   1:  PR[91,3] = PR[90,3] + 65.195;
   1:L PR[91] R[100]mm/sec CNT100;
   1:  PR[91,1] = PR[90,1] + -66.038;
   1:  PR[91,2] = PR[90,2] + 18.167;
   1:  PR[91,3] = PR[90,3] + 63.911;
   1:L PR[91] R[100]mm/sec CNT100;
   1:  PR[91,1] = PR[90,1] + -70.511;
   1:  PR[91,2] = PR[90,2] + 15.205;
   1:L PR[91] R[100]mm/sec CNT100;
   1:  PR[91,1] = PR[90,1] + -74.081;
   1:  PR[91,2] = PR[90,2] + 11.663;
   1:  PR[91,3] = PR[90,3] + 63.930;
   1:L PR[91] R[100]mm/sec CNT100;
   1:  PR[91,1] = PR[90,1] + -76.653;
   1:  PR[91,2] = PR[90,2] + 7.733;
   1:  PR[91,3] = PR[90,3] + 63.947;
   1:L PR[91] R[100]mm/sec CNT100;
   1:  PR[91,1] = PR[90,1] + -78.198;
   1:  PR[91,2] = PR[90,2] + 3.559;
   1:  PR[91,3] = PR[90,3] + 63.964;
   1:L PR[91] R[100]mm/sec CNT100;
   1:  PR[91,1] = PR[90,1] + -78.594;
   1:  PR[91,2] = PR[90,2] + 0.279;
   1:  PR[91,3] = PR[90,3] + 63.979;
   1:L PR[91] R[100]mm/sec CNT100;
   1:  PR[91,1] = PR[90,1] + -78.770;
   1:  PR[91,2] = PR[90,2] + -0.700;
   1:  PR[91,3] = PR[90,3] + 63.991;
   1:L PR[91] R[100]mm/sec CNT100;
   1:  PR[91,1] = PR[90,1] + -78.578;
   1:  PR[91,2] = PR[90,2] + -1.617;
   1:  PR[91,3] = PR[90,3] + 63.994;
   1:L PR[91] R[100]mm/sec CNT100;
   1:  PR[91,1] = PR[90,1] + -78.140;
   1:  PR[91,2] = PR[90,2] + -5.208;
   1:  PR[91,3] = PR[90,3] + 63.998;
   1:L PR[91] R[100]mm/sec CNT100;
   1:  PR[91,1] = PR[90,1] + -77.858;
   1:  PR[91,2] = PR[90,2] + -5.991;
   1:  PR[91,3] = PR[90,3] + 64.010;
   1:L PR[91] R[100]mm/sec CNT100;
   1:  PR[91,1] = PR[90,1] + -76.508;
   1:  PR[91,2] = PR[90,2] + -9.566;
   1:  PR[91,3] = PR[90,3] + 64.013;
   1:L PR[91] R[100]mm/sec CNT100;
   1:  PR[91,1] = PR[90,1] + -76.251;
   1:  PR[91,2] = PR[90,2] + -9.971;
   1:  PR[91,3] = PR[90,3] + 64.027;
   1:L PR[91] R[100]mm/sec CNT100;
   1:  PR[91,1] = PR[90,1] + -73.777;
   1:  PR[91,2] = PR[90,2] + -13.651;
   1:  PR[91,3] = PR[90,3] + 64.028;
   1:L PR[91] R[100]mm/sec CNT100;
   1:  PR[91,1] = PR[90,1] + -73.531;
   1:  PR[91,2] = PR[90,2] + -13.889;
   1:  PR[91,3] = PR[90,3] + 64.044;
   1:L PR[91] R[100]mm/sec CNT100;
   1:  PR[91,1] = PR[90,1] + -69.827;
   1:  PR[91,2] = PR[90,2] + -17.193;
   1:  PR[91,3] = PR[90,3] + 64.045;
   1:L PR[91] R[100]mm/sec CNT100;
   1:  PR[91,1] = PR[90,1] + -68.494;
   1:  PR[91,2] = PR[90,2] + -17.992;
   1:  PR[91,3] = PR[90,3] + 64.062;
   1:L PR[91] R[100]mm/sec CNT100;
   1:  PR[91,1] = PR[90,1] + -64.853;
   1:  PR[91,2] = PR[90,2] + -20.132;
   1:  PR[91,3] = PR[90,3] + 64.068;
   1:L PR[91] R[100]mm/sec CNT100;
   1:  PR[91,1] = PR[90,1] + -60.373;
   1:  PR[91,2] = PR[90,2] + -21.812;
   1:  PR[91,3] = PR[90,3] + 64.083;
   1:L PR[91] R[100]mm/sec CNT100;
   1:  PR[91,1] = PR[90,1] + -59.088;
   1:  PR[91,2] = PR[90,2] + -22.281;
   1:  PR[91,3] = PR[90,3] + 64.099;
   1:L PR[91] R[100]mm/sec CNT100;
   1:  PR[91,1] = PR[90,1] + -52.980;
   1:  PR[91,2] = PR[90,2] + -23.447;
   1:  PR[91,3] = PR[90,3] + 64.104;
   1:L PR[91] R[100]mm/sec CNT100;
   1:  PR[91,1] = PR[90,1] + -50.323;
   1:  PR[91,2] = PR[90,2] + -23.702;
   1:  PR[91,3] = PR[90,3] + 64.126;
   1:L PR[91] R[100]mm/sec CNT100;
   1:  PR[91,1] = PR[90,1] + -47.192;
   1:  PR[91,2] = PR[90,2] + -23.829;
   1:  PR[91,3] = PR[90,3] + 64.135;
   1:L PR[91] R[100]mm/sec CNT100;
   1:  PR[91,1] = PR[90,1] + -43.588;
   1:  PR[91,2] = PR[90,2] + -23.669;
   1:  PR[91,3] = PR[90,3] + 64.146;
   1:L PR[91] R[100]mm/sec CNT100;
   1:  PR[91,1] = PR[90,1] + -41.498;
   1:  PR[91,2] = PR[90,2] + -23.638;
   1:  PR[91,3] = PR[90,3] + 64.159;
   1:L PR[91] R[100]mm/sec CNT100;
   1:  PR[91,1] = PR[90,1] + -39.473;
   1:  PR[91,2] = PR[90,2] + -23.516;
   1:  PR[91,3] = PR[90,3] + 64.166;
   1:L PR[91] R[100]mm/sec CNT100;
   1:  PR[91,1] = PR[90,1] + -36.086;
   1:  PR[91,2] = PR[90,2] + -23.043;
   1:  PR[91,3] = PR[90,3] + 64.173;
   1:L PR[91] R[100]mm/sec CNT100;
   1:  PR[91,1] = PR[90,1] + -32.879;
   1:  PR[91,2] = PR[90,2] + -22.411;
   1:  PR[91,3] = PR[90,3] + 64.185;
   1:L PR[91] R[100]mm/sec CNT100;
   1:  PR[91,1] = PR[90,1] + -29.442;
   1:  PR[91,2] = PR[90,2] + -21.943;
   1:  PR[91,3] = PR[90,3] + 64.197;
   1:L PR[91] R[100]mm/sec CNT100;
   1:  PR[91,1] = PR[90,1] + -23.128;
   1:  PR[91,2] = PR[90,2] + -20.482;
   1:  PR[91,3] = PR[90,3] + 64.209;
   1:L PR[91] R[100]mm/sec CNT100;
   1:  PR[91,1] = PR[90,1] + -19.496;
   1:  PR[91,2] = PR[90,2] + -22.048;
   1:  PR[91,3] = PR[90,3] + 64.231;
   1:L PR[91] R[100]mm/sec CNT100;
   1:  PR[91,1] = PR[90,1] + -17.322;
   1:  PR[91,2] = PR[90,2] + -22.682;
   1:  PR[91,3] = PR[90,3] + 64.245;
   1:L PR[91] R[100]mm/sec CNT100;
   1:  PR[91,1] = PR[90,1] + -14.113;
   1:  PR[91,2] = PR[90,2] + -23.536;
   1:  PR[91,3] = PR[90,3] + 64.253;
   1:L PR[91] R[100]mm/sec CNT100;
   1:  PR[91,1] = PR[90,1] + -8.398;
   1:  PR[91,2] = PR[90,2] + -23.980;
   1:  PR[91,3] = PR[90,3] + 64.265;
   1:L PR[91] R[100]mm/sec CNT100;
   1:  PR[91,1] = PR[90,1] + -2.492;
   1:  PR[91,2] = PR[90,2] + -23.372;
   1:  PR[91,3] = PR[90,3] + 64.285;
   1:L PR[91] R[100]mm/sec CNT100;
   1:  PR[91,1] = PR[90,1] + -0.519;
   1:  PR[91,2] = PR[90,2] + -22.811;
   1:  PR[91,3] = PR[90,3] + 64.306;
   1:L PR[91] R[100]mm/sec CNT100;
   1:  PR[91,1] = PR[90,1] + 3.330;
   1:  PR[91,2] = PR[90,2] + -21.668;
   1:  PR[91,3] = PR[90,3] + 64.313;
   1:L PR[91] R[100]mm/sec CNT100;
   1:  PR[91,1] = PR[90,1] + 6.156;
   1:  PR[91,2] = PR[90,2] + -20.297;
   1:  PR[91,3] = PR[90,3] + 64.327;
   1:L PR[91] R[100]mm/sec CNT100;
   1:  PR[91,1] = PR[90,1] + 11.934;
   1:  PR[91,2] = PR[90,2] + -23.385;
   1:  PR[91,3] = PR[90,3] + 64.338;
   1:L PR[91] R[100]mm/sec CNT100;
   1:  PR[91,1] = PR[90,1] + 17.314;
   1:  PR[91,2] = PR[90,2] + -24.854;
   1:  PR[91,3] = PR[90,3] + 64.361;
   1:L PR[91] R[100]mm/sec CNT100;
   1:  PR[91,1] = PR[90,1] + 22.909;
   1:  PR[91,2] = PR[90,2] + -25.082;
   1:  PR[91,3] = PR[90,3] + 64.380;
   1:L PR[91] R[100]mm/sec CNT100;
   1:  PR[91,1] = PR[90,1] + 28.505;
   1:  PR[91,2] = PR[90,2] + -24.027;
   1:  PR[91,3] = PR[90,3] + 64.400;
   1:L PR[91] R[100]mm/sec CNT100;
   1:  PR[91,1] = PR[90,1] + 29.696;
   1:  PR[91,2] = PR[90,2] + -23.650;
   1:  PR[91,3] = PR[90,3] + 64.420;
   1:L PR[91] R[100]mm/sec CNT100;
   1:  PR[91,1] = PR[90,1] + 33.478;
   1:  PR[91,2] = PR[90,2] + -24.727;
   1:  PR[91,3] = PR[90,3] + 64.424;
   1:L PR[91] R[100]mm/sec CNT100;
   1:  PR[91,1] = PR[90,1] + 35.307;
   1:  PR[91,2] = PR[90,2] + -25.218;
   1:  PR[91,3] = PR[90,3] + 64.438;
   1:L PR[91] R[100]mm/sec CNT100;
   1:  PR[91,1] = PR[90,1] + 41.330;
   1:  PR[91,2] = PR[90,2] + -25.987;
   1:  PR[91,3] = PR[90,3] + 64.445;
   1:L PR[91] R[100]mm/sec CNT100;
   1:  PR[91,1] = PR[90,1] + 45.575;
   1:  PR[91,2] = PR[90,2] + -26.004;
   1:  PR[91,3] = PR[90,3] + 64.466;
   1:L PR[91] R[100]mm/sec CNT100;
   1:  PR[91,1] = PR[90,1] + 46.620;
   1:  PR[91,2] = PR[90,2] + -26.023;
   1:  PR[91,3] = PR[90,3] + 64.481;
   1:L PR[91] R[100]mm/sec CNT100;
   1:  PR[91,1] = PR[90,1] + 49.214;
   1:  PR[91,2] = PR[90,2] + -25.837;
   1:  PR[91,3] = PR[90,3] + 64.485;
   1:L PR[91] R[100]mm/sec CNT100;
   1:  PR[91,1] = PR[90,1] + 51.095;
   1:  PR[91,2] = PR[90,2] + -25.664;
   1:  PR[91,3] = PR[90,3] + 64.494;
   1:L PR[91] R[100]mm/sec CNT100;
   1:  PR[91,1] = PR[90,1] + 56.435;
   1:  PR[91,2] = PR[90,2] + -24.677;
   1:  PR[91,3] = PR[90,3] + 64.500;
   1:L PR[91] R[100]mm/sec CNT100;
   1:  PR[91,1] = PR[90,1] + 63.147;
   1:  PR[91,2] = PR[90,2] + -22.494;
   1:  PR[91,3] = PR[90,3] + 64.519;
   1:L PR[91] R[100]mm/sec CNT100;
   1:  PR[91,1] = PR[90,1] + 63.555;
   1:  PR[91,2] = PR[90,2] + -22.305;
   1:  PR[91,3] = PR[90,3] + 64.544;
   1:L PR[91] R[100]mm/sec CNT100;
   1:  PR[91,1] = PR[90,1] + 65.028;
   1:  PR[91,2] = PR[90,2] + -21.507;
   1:  PR[91,3] = PR[90,3] + 64.546;
   1:L PR[91] R[100]mm/sec CNT100;
   1:  PR[91,1] = PR[90,1] + 69.095;
   1:  PR[91,2] = PR[90,2] + -19.132;
   1:  PR[91,3] = PR[90,3] + 64.551;
   1:L PR[91] R[100]mm/sec CNT100;
   1:  PR[91,1] = PR[90,1] + 71.773;
   1:  PR[91,2] = PR[90,2] + -16.745;
   1:  PR[91,3] = PR[90,3] + 64.568;
   1:L PR[91] R[100]mm/sec CNT100;
   1:  PR[91,1] = PR[90,1] + 73.617;
   1:  PR[91,2] = PR[90,2] + -15.079;
   1:  PR[91,3] = PR[90,3] + 64.580;
   1:L PR[91] R[100]mm/sec CNT100;
   1:  PR[91,1] = PR[90,1] + 76.861;
   1:  PR[91,2] = PR[90,2] + -10.536;
   1:  PR[91,3] = PR[90,3] + 64.589;
   1:L PR[91] R[100]mm/sec CNT100;
   1:  PR[91,1] = PR[90,1] + 78.802;
   1:  PR[91,2] = PR[90,2] + -5.697;
   1:  PR[91,3] = PR[90,3] + 64.609;
   1:L PR[91] R[100]mm/sec CNT100;
   1:  PR[91,1] = PR[90,1] + 79.399;
   1:  PR[91,2] = PR[90,2] + -1.168;
   1:  PR[91,3] = PR[90,3] + 64.627;
   1:L PR[91] R[100]mm/sec CNT100;
   1:  PR[91,1] = PR[90,1] + 79.474;
   1:  PR[91,2] = PR[90,2] + -0.700;
   1:  PR[91,3] = PR[90,3] + 64.643;
   1:L PR[91] R[100]mm/sec CNT100;
   1:  PR[91,1] = PR[90,1] + 78.963;
   1:  PR[91,2] = PR[90,2] + 3.215;
   1:  PR[91,3] = PR[90,3] + 64.645;
   1:L PR[91] R[100]mm/sec CNT100;
   1:  PR[91,1] = PR[90,1] + 78.903;
   1:  PR[91,2] = PR[90,2] + 3.455;
   1:  PR[91,3] = PR[90,3] + 64.658;
   1:L PR[91] R[100]mm/sec CNT100;
   1:  PR[91,1] = PR[90,1] + 78.799;
   1:  PR[91,2] = PR[90,2] + 4.246;
   1:  PR[91,3] = PR[90,3] + 64.659;
   1:L PR[91] R[100]mm/sec CNT100;
   1:  PR[91,1] = PR[90,1] + 76.856;
   1:  PR[91,2] = PR[90,2] + 9.086;
   1:  PR[91,3] = PR[90,3] + 64.662;
   1:L PR[91] R[100]mm/sec CNT100;
   1:  PR[91,1] = PR[90,1] + 73.613;
   1:  PR[91,2] = PR[90,2] + 13.624;
   1:  PR[91,3] = PR[90,3] + 64.680;
   1:L PR[91] R[100]mm/sec CNT100;
   1:  PR[91,1] = PR[90,1] + 69.094;
   1:  PR[91,2] = PR[90,2] + 17.673;
   1:  PR[91,3] = PR[90,3] + 64.700;
   1:L PR[91] R[100]mm/sec CNT100;
   1:  PR[91,1] = PR[90,1] + 65.028;
   1:  PR[91,2] = PR[90,2] + 20.050;
   1:  PR[91,3] = PR[90,3] + 64.721;
   1:L PR[91] R[100]mm/sec CNT100;
   1:  PR[91,1] = PR[90,1] + 63.571;
   1:  PR[91,2] = PR[90,2] + 20.840;
   1:  PR[91,3] = PR[90,3] + 64.738;
   1:L PR[91] R[100]mm/sec CNT100;
   1:  PR[91,1] = PR[90,1] + 63.168;
   1:  PR[91,2] = PR[90,2] + 21.026;
   1:  PR[91,3] = PR[90,3] + 64.743;
   1:L PR[91] R[100]mm/sec CNT100;
   1:  PR[91,1] = PR[90,1] + 56.445;
   1:  PR[91,2] = PR[90,2] + 23.216;
   1:  PR[91,3] = PR[90,3] + 64.745;
   1:L PR[91] R[100]mm/sec CNT100;
   1:  PR[91,1] = PR[90,1] + 51.095;
   1:  PR[91,2] = PR[90,2] + 24.206;
   1:  PR[91,3] = PR[90,3] + 64.770;
   1:L PR[91] R[100]mm/sec CNT100;
   1:  PR[91,1] = PR[90,1] + 49.215;
   1:  PR[91,2] = PR[90,2] + 24.378;
   1:  PR[91,3] = PR[90,3] + 64.789;
   1:L PR[91] R[100]mm/sec CNT100;
   1:  PR[91,1] = PR[90,1] + 46.620;
   1:  PR[91,2] = PR[90,2] + 24.564;
   1:  PR[91,3] = PR[90,3] + 64.795;
   1:L PR[91] R[100]mm/sec CNT100;
   1:  PR[91,1] = PR[90,1] + 45.575;
   1:  PR[91,2] = PR[90,2] + 24.545;
   1:  PR[91,3] = PR[90,3] + 64.804;
   1:L PR[91] R[100]mm/sec CNT100;
   1:  PR[91,1] = PR[90,1] + 41.330;
   1:  PR[91,2] = PR[90,2] + 24.528;
   1:  PR[91,3] = PR[90,3] + 64.808;
   1:L PR[91] R[100]mm/sec CNT100;
   1:  PR[91,1] = PR[90,1] + 35.307;
   1:  PR[91,2] = PR[90,2] + 23.759;
   1:  PR[91,3] = PR[90,3] + 64.823;
   1:L PR[91] R[100]mm/sec CNT100;
   1:  PR[91,1] = PR[90,1] + 33.478;
   1:  PR[91,2] = PR[90,2] + 23.268;
   1:  PR[91,3] = PR[90,3] + 64.844;
   1:L PR[91] R[100]mm/sec CNT100;
   1:  PR[91,1] = PR[90,1] + 29.686;
   1:  PR[91,2] = PR[90,2] + 22.188;
   1:  PR[91,3] = PR[90,3] + 64.851;
   1:L PR[91] R[100]mm/sec CNT100;
   1:  PR[91,1] = PR[90,1] + 28.655;
   1:  PR[91,2] = PR[90,2] + 22.526;
   1:  PR[91,3] = PR[90,3] + 64.865;
   1:L PR[91] R[100]mm/sec CNT100;
   1:  PR[91,1] = PR[90,1] + 27.759;
   1:  PR[91,2] = PR[90,2] + 22.715;
   1:  PR[91,3] = PR[90,3] + 64.868;
   1:L PR[91] R[100]mm/sec CNT100;
   1:  PR[91,1] = PR[90,1] + 22.910;
   1:  PR[91,2] = PR[90,2] + 23.623;
   1:  PR[91,3] = PR[90,3] + 64.872;
   1:L PR[91] R[100]mm/sec CNT100;
   1:  PR[91,1] = PR[90,1] + 17.313;
   1:  PR[91,2] = PR[90,2] + 23.395;
   1:  PR[91,3] = PR[90,3] + 64.889;
   1:L PR[91] R[100]mm/sec CNT100;
   1:  PR[91,1] = PR[90,1] + 11.931;
   1:  PR[91,2] = PR[90,2] + 21.925;
   1:  PR[91,3] = PR[90,3] + 64.909;
   1:L PR[91] R[100]mm/sec CNT100;
   1:  PR[91,1] = PR[90,1] + 6.142;
   1:  PR[91,2] = PR[90,2] + 18.842;
   1:  PR[91,3] = PR[90,3] + 64.928;
   1:L PR[91] R[100]mm/sec CNT100;
   1:  PR[91,1] = PR[90,1] + 4.093;
   1:  PR[91,2] = PR[90,2] + 19.856;
   1:  PR[91,3] = PR[90,3] + 64.951;
   1:L PR[91] R[100]mm/sec CNT100;
   1:  PR[91,1] = PR[90,1] + 3.348;
   1:  PR[91,2] = PR[90,2] + 20.203;
   1:  PR[91,3] = PR[90,3] + 64.959;
   1:L PR[91] R[100]mm/sec CNT100;
   1:  PR[91,1] = PR[90,1] + -0.515;
   1:  PR[91,2] = PR[90,2] + 21.353;
   1:  PR[91,3] = PR[90,3] + 64.962;
   1:L PR[91] R[100]mm/sec CNT100;
   1:  PR[91,1] = PR[90,1] + -2.470;
   1:  PR[91,2] = PR[90,2] + 21.909;
   1:  PR[91,3] = PR[90,3] + 64.976;
   1:L PR[91] R[100]mm/sec CNT100;
   1:  PR[91,1] = PR[90,1] + -8.387;
   1:  PR[91,2] = PR[90,2] + 22.521;
   1:  PR[91,3] = PR[90,3] + 64.983;
   1:L PR[91] R[100]mm/sec CNT100;
   1:  PR[91,1] = PR[90,1] + -14.097;
   1:  PR[91,2] = PR[90,2] + 22.080;
   1:  PR[91,3] = PR[90,3] + 65.004;
   1:L PR[91] R[100]mm/sec CNT100;
   1:  PR[91,1] = PR[90,1] + -17.311;
   1:  PR[91,2] = PR[90,2] + 21.224;
   1:  PR[91,3] = PR[90,3] + 65.024;
   1:L PR[91] R[100]mm/sec CNT100;
   1:  PR[91,1] = PR[90,1] + -19.480;
   1:  PR[91,2] = PR[90,2] + 20.596;
   1:  PR[91,3] = PR[90,3] + 65.036;
   1:L PR[91] R[100]mm/sec CNT100;
   1:  PR[91,1] = PR[90,1] + -23.127;
   1:  PR[91,2] = PR[90,2] + 19.024;
   1:  PR[91,3] = PR[90,3] + 65.044;
   1:L PR[91] R[100]mm/sec CNT100;
   1:  PR[91,1] = PR[90,1] + -29.591;
   1:  PR[91,2] = PR[90,2] + 20.509;
   1:  PR[91,3] = PR[90,3] + 65.057;
   1:L PR[91] R[100]mm/sec CNT100;
   1:  PR[91,1] = PR[90,1] + -31.869;
   1:  PR[91,2] = PR[90,2] + 20.801;
   1:  PR[91,3] = PR[90,3] + 65.081;
   1:L PR[91] R[100]mm/sec CNT100;
   1:  PR[91,1] = PR[90,1] + -36.385;
   1:  PR[91,2] = PR[90,2] + 21.658;
   1:  PR[91,3] = PR[90,3] + 65.089;
   1:L PR[91] R[100]mm/sec CNT100;
   1:  PR[91,1] = PR[90,1] + -41.380;
   1:  PR[91,2] = PR[90,2] + 22.076;
   1:  PR[91,3] = PR[90,3] + 65.105;
   1:L PR[91] R[100]mm/sec CNT100;
   1:  PR[91,1] = PR[90,1] + -42.819;
   1:  PR[91,2] = PR[90,2] + 22.268;
   1:  PR[91,3] = PR[90,3] + 65.122;
   1:L PR[91] R[100]mm/sec CNT100;
   1:  PR[91,1] = PR[90,1] + -44.055;
   1:  PR[91,2] = PR[90,2] + 22.365;
   1:  PR[91,3] = PR[90,3] + 65.127;
   1:L PR[91] R[100]mm/sec CNT100;
   1:  PR[91,1] = PR[90,1] + -47.939;
   1:  PR[91,2] = PR[90,2] + 22.299;
   1:  PR[91,3] = PR[90,3] + 65.132;
   1:L PR[91] R[100]mm/sec CNT100;
   1:  PR[91,1] = PR[90,1] + -53.378;
   1:  PR[91,2] = PR[90,2] + 21.968;
   1:  PR[91,3] = PR[90,3] + 65.145;
   1:L PR[91] R[100]mm/sec CNT100;
   1:  PR[91,1] = PR[90,1] + -57.549;
   1:  PR[91,2] = PR[90,2] + 21.084;
   1:  PR[91,3] = PR[90,3] + 65.164;
   1:L PR[91] R[100]mm/sec CNT100;
   1:  PR[91,1] = PR[90,1] + -60.125;
   1:  PR[91,2] = PR[90,2] + 20.512;
   1:  PR[91,3] = PR[90,3] + 65.179;
   1:L PR[91] R[100]mm/sec CNT100;
   1:  PR[91,1] = PR[90,1] + -61.822;
   1:  PR[91,2] = PR[90,2] + 19.851;
   1:  PR[91,3] = PR[90,3] + 65.189;
   1:L PR[91] R[100]mm/sec CNT100;
   1:  PR[91] = PR[90];
   1:  PR[91,1] = PR[90,1] + -64.918;
   1:  PR[91,2] = PR[90,2] + 18.355;
   1:  PR[91,3] = PR[90,3] + 66.495;
   1:L PR[91] R[100]mm/sec CNT100;
   1:  PR[91,1] = PR[90,1] + -67.688;
   1:  PR[91,2] = PR[90,2] + 16.655;
   1:  PR[91,3] = PR[90,3] + 65.208;
   1:L PR[91] R[100]mm/sec CNT100;
   1:  PR[91,1] = PR[90,1] + -69.669;
   1:  PR[91,2] = PR[90,2] + 15.342;
   1:  PR[91,3] = PR[90,3] + 65.220;
   1:L PR[91] R[100]mm/sec CNT100;
   1:  PR[91,1] = PR[90,1] + -73.276;
   1:  PR[91,2] = PR[90,2] + 11.769;
   1:  PR[91,3] = PR[90,3] + 65.228;
   1:L PR[91] R[100]mm/sec CNT100;
   1:  PR[91,1] = PR[90,1] + -75.873;
   1:  PR[91,2] = PR[90,2] + 7.805;
   1:  PR[91,3] = PR[90,3] + 65.246;
   1:L PR[91] R[100]mm/sec CNT100;
   1:  PR[91,1] = PR[90,1] + -77.433;
   1:  PR[91,2] = PR[90,2] + 3.596;
   1:  PR[91,3] = PR[90,3] + 65.263;
   1:L PR[91] R[100]mm/sec CNT100;
   1:  PR[91,1] = PR[90,1] + -77.752;
   1:  PR[91,2] = PR[90,2] + 0.956;
   1:  PR[91,3] = PR[90,3] + 65.279;
   1:L PR[91] R[100]mm/sec CNT100;
   1:  PR[91,1] = PR[90,1] + -78.050;
   1:  PR[91,2] = PR[90,2] + -0.700;
   1:  PR[91,3] = PR[90,3] + 65.288;
   1:L PR[91] R[100]mm/sec CNT100;
   1:  PR[91,1] = PR[90,1] + -77.966;
   1:  PR[91,2] = PR[90,2] + -1.098;
   1:  PR[91,3] = PR[90,3] + 65.294;
   1:L PR[91] R[100]mm/sec CNT100;
   1:  PR[91,1] = PR[90,1] + -77.460;
   1:  PR[91,2] = PR[90,2] + -5.248;
   1:  PR[91,3] = PR[90,3] + 65.295;
   1:L PR[91] R[100]mm/sec CNT100;
   1:  PR[91,1] = PR[90,1] + -75.804;
   1:  PR[91,2] = PR[90,2] + -9.653;
   1:  PR[91,3] = PR[90,3] + 65.310;
   1:L PR[91] R[100]mm/sec CNT100;
   1:  PR[91,1] = PR[90,1] + -75.073;
   1:  PR[91,2] = PR[90,2] + -10.749;
   1:  PR[91,3] = PR[90,3] + 65.327;
   1:L PR[91] R[100]mm/sec CNT100;
   1:  PR[91,1] = PR[90,1] + -72.949;
   1:  PR[91,2] = PR[90,2] + -13.691;
   1:  PR[91,3] = PR[90,3] + 65.331;
   1:L PR[91] R[100]mm/sec CNT100;
   1:  PR[91,1] = PR[90,1] + -68.910;
   1:  PR[91,2] = PR[90,2] + -17.302;
   1:  PR[91,3] = PR[90,3] + 65.344;
   1:L PR[91] R[100]mm/sec CNT100;
   1:  PR[91,1] = PR[90,1] + -66.512;
   1:  PR[91,2] = PR[90,2] + -18.739;
   1:  PR[91,3] = PR[90,3] + 65.363;
   1:L PR[91] R[100]mm/sec CNT100;
   1:  PR[91,1] = PR[90,1] + -63.913;
   1:  PR[91,2] = PR[90,2] + -20.268;
   1:  PR[91,3] = PR[90,3] + 65.373;
   1:L PR[91] R[100]mm/sec CNT100;
   1:  PR[91,1] = PR[90,1] + -58.107;
   1:  PR[91,2] = PR[90,2] + -22.444;
   1:  PR[91,3] = PR[90,3] + 65.384;
   1:L PR[91] R[100]mm/sec CNT100;
   1:  PR[91,1] = PR[90,1] + -52.157;
   1:  PR[91,2] = PR[90,2] + -23.581;
   1:  PR[91,3] = PR[90,3] + 65.406;
   1:L PR[91] R[100]mm/sec CNT100;
   1:  PR[91,1] = PR[90,1] + -47.855;
   1:  PR[91,2] = PR[90,2] + -23.994;
   1:  PR[91,3] = PR[90,3] + 65.427;
   1:L PR[91] R[100]mm/sec CNT100;
   1:  PR[91,1] = PR[90,1] + -46.414;
   1:  PR[91,2] = PR[90,2] + -24.052;
   1:  PR[91,3] = PR[90,3] + 65.443;
   1:L PR[91] R[100]mm/sec CNT100;
   1:  PR[91,1] = PR[90,1] + -44.701;
   1:  PR[91,2] = PR[90,2] + -23.976;
   1:  PR[91,3] = PR[90,3] + 65.448;
   1:L PR[91] R[100]mm/sec CNT100;
   1:  PR[91,1] = PR[90,1] + -40.730;
   1:  PR[91,2] = PR[90,2] + -23.917;
   1:  PR[91,3] = PR[90,3] + 65.454;
   1:L PR[91] R[100]mm/sec CNT100;
   1:  PR[91,1] = PR[90,1] + -36.785;
   1:  PR[91,2] = PR[90,2] + -23.680;
   1:  PR[91,3] = PR[90,3] + 65.468;
   1:L PR[91] R[100]mm/sec CNT100;
   1:  PR[91,1] = PR[90,1] + -35.256;
   1:  PR[91,2] = PR[90,2] + -23.467;
   1:  PR[91,3] = PR[90,3] + 65.482;
   1:L PR[91] R[100]mm/sec CNT100;
   1:  PR[91,1] = PR[90,1] + -33.740;
   1:  PR[91,2] = PR[90,2] + -23.168;
   1:  PR[91,3] = PR[90,3] + 65.487;
   1:L PR[91] R[100]mm/sec CNT100;
   1:  PR[91,1] = PR[90,1] + -27.820;
   1:  PR[91,2] = PR[90,2] + -22.362;
   1:  PR[91,3] = PR[90,3] + 65.493;
   1:L PR[91] R[100]mm/sec CNT100;
   1:  PR[91,1] = PR[90,1] + -24.290;
   1:  PR[91,2] = PR[90,2] + -21.549;
   1:  PR[91,3] = PR[90,3] + 65.514;
   1:L PR[91] R[100]mm/sec CNT100;
   1:  PR[91,1] = PR[90,1] + -21.649;
   1:  PR[91,2] = PR[90,2] + -21.053;
   1:  PR[91,3] = PR[90,3] + 65.526;
   1:L PR[91] R[100]mm/sec CNT100;
   1:  PR[91,1] = PR[90,1] + -18.816;
   1:  PR[91,2] = PR[90,2] + -22.269;
   1:  PR[91,3] = PR[90,3] + 65.536;
   1:L PR[91] R[100]mm/sec CNT100;
   1:  PR[91,1] = PR[90,1] + -17.201;
   1:  PR[91,2] = PR[90,2] + -22.739;
   1:  PR[91,3] = PR[90,3] + 65.547;
   1:L PR[91] R[100]mm/sec CNT100;
   1:  PR[91,1] = PR[90,1] + -13.448;
   1:  PR[91,2] = PR[90,2] + -23.739;
   1:  PR[91,3] = PR[90,3] + 65.553;
   1:L PR[91] R[100]mm/sec CNT100;
   1:  PR[91,1] = PR[90,1] + -7.645;
   1:  PR[91,2] = PR[90,2] + -24.196;
   1:  PR[91,3] = PR[90,3] + 65.567;
   1:L PR[91] R[100]mm/sec CNT100;
   1:  PR[91,1] = PR[90,1] + -6.885;
   1:  PR[91,2] = PR[90,2] + -24.130;
   1:  PR[91,3] = PR[90,3] + 65.587;
   1:L PR[91] R[100]mm/sec CNT100;
   1:  PR[91,1] = PR[90,1] + -1.660;
   1:  PR[91,2] = PR[90,2] + -23.602;
   1:  PR[91,3] = PR[90,3] + 65.590;
   1:L PR[91] R[100]mm/sec CNT100;
   1:  PR[91,1] = PR[90,1] + 1.593;
   1:  PR[91,2] = PR[90,2] + -22.676;
   1:  PR[91,3] = PR[90,3] + 65.608;
   1:L PR[91] R[100]mm/sec CNT100;
   1:  PR[91,1] = PR[90,1] + 4.238;
   1:  PR[91,2] = PR[90,2] + -21.891;
   1:  PR[91,3] = PR[90,3] + 65.620;
   1:L PR[91] R[100]mm/sec CNT100;
   1:  PR[91,1] = PR[90,1] + 6.446;
   1:  PR[91,2] = PR[90,2] + -20.820;
   1:  PR[91,3] = PR[90,3] + 65.630;
   1:L PR[91] R[100]mm/sec CNT100;
   1:  PR[91,1] = PR[90,1] + 10.926;
   1:  PR[91,2] = PR[90,2] + -23.208;
   1:  PR[91,3] = PR[90,3] + 65.639;
   1:L PR[91] R[100]mm/sec CNT100;
   1:  PR[91,1] = PR[90,1] + 11.742;
   1:  PR[91,2] = PR[90,2] + -23.583;
   1:  PR[91,3] = PR[90,3] + 65.657;
   1:L PR[91] R[100]mm/sec CNT100;
   1:  PR[91,1] = PR[90,1] + 17.142;
   1:  PR[91,2] = PR[90,2] + -25.054;
   1:  PR[91,3] = PR[90,3] + 65.660;
   1:L PR[91] R[100]mm/sec CNT100;
   1:  PR[91,1] = PR[90,1] + 17.170;
   1:  PR[91,2] = PR[90,2] + -25.060;
   1:  PR[91,3] = PR[90,3] + 65.680;
   1:L PR[91] R[100]mm/sec CNT100;
   1:  PR[91,1] = PR[90,1] + 22.787;
   1:  PR[91,2] = PR[90,2] + -25.287;
   1:L PR[91] R[100]mm/sec CNT100;
   1:  PR[91,1] = PR[90,1] + 28.397;
   1:  PR[91,2] = PR[90,2] + -24.234;
   1:  PR[91,3] = PR[90,3] + 65.700;
   1:L PR[91] R[100]mm/sec CNT100;
   1:  PR[91,1] = PR[90,1] + 29.133;
   1:  PR[91,2] = PR[90,2] + -24.016;
   1:  PR[91,3] = PR[90,3] + 65.720;
   1:L PR[91] R[100]mm/sec CNT100;
   1:  PR[91,1] = PR[90,1] + 32.821;
   1:  PR[91,2] = PR[90,2] + -25.060;
   1:  PR[91,3] = PR[90,3] + 65.722;
   1:L PR[91] R[100]mm/sec CNT100;
   1:  PR[91,1] = PR[90,1] + 34.276;
   1:  PR[91,2] = PR[90,2] + -25.447;
   1:  PR[91,3] = PR[90,3] + 65.736;
   1:L PR[91] R[100]mm/sec CNT100;
   1:  PR[91,1] = PR[90,1] + 40.204;
   1:  PR[91,2] = PR[90,2] + -26.207;
   1:  PR[91,3] = PR[90,3] + 65.741;
   1:L PR[91] R[100]mm/sec CNT100;
   1:  PR[91,1] = PR[90,1] + 45.797;
   1:  PR[91,2] = PR[90,2] + -26.222;
   1:  PR[91,3] = PR[90,3] + 65.762;
   1:L PR[91] R[100]mm/sec CNT100;
   1:  PR[91,1] = PR[90,1] + 46.538;
   1:  PR[91,2] = PR[90,2] + -26.133;
   1:  PR[91,3] = PR[90,3] + 65.782;
   1:L PR[91] R[100]mm/sec CNT100;
   1:  PR[91,1] = PR[90,1] + 50.425;
   1:  PR[91,2] = PR[90,2] + -25.777;
   1:  PR[91,3] = PR[90,3] + 65.785;
   1:L PR[91] R[100]mm/sec CNT100;
   1:  PR[91,1] = PR[90,1] + 55.385;
   1:  PR[91,2] = PR[90,2] + -24.854;
   1:  PR[91,3] = PR[90,3] + 65.799;
   1:L PR[91] R[100]mm/sec CNT100;
   1:  PR[91,1] = PR[90,1] + 61.784;
   1:  PR[91,2] = PR[90,2] + -22.774;
   1:  PR[91,3] = PR[90,3] + 65.816;
   1:L PR[91] R[100]mm/sec CNT100;
   1:  PR[91,1] = PR[90,1] + 62.965;
   1:  PR[91,2] = PR[90,2] + -22.228;
   1:  PR[91,3] = PR[90,3] + 65.840;
   1:L PR[91] R[100]mm/sec CNT100;
   1:  PR[91,1] = PR[90,1] + 66.536;
   1:  PR[91,2] = PR[90,2] + -20.295;
   1:  PR[91,3] = PR[90,3] + 65.845;
   1:L PR[91] R[100]mm/sec CNT100;
   1:  PR[91,1] = PR[90,1] + 68.202;
   1:  PR[91,2] = PR[90,2] + -19.322;
   1:  PR[91,3] = PR[90,3] + 65.859;
   1:L PR[91] R[100]mm/sec CNT100;
   1:  PR[91,1] = PR[90,1] + 72.782;
   1:  PR[91,2] = PR[90,2] + -15.222;
   1:  PR[91,3] = PR[90,3] + 65.866;
   1:L PR[91] R[100]mm/sec CNT100;
   1:  PR[91,1] = PR[90,1] + 76.061;
   1:  PR[91,2] = PR[90,2] + -10.636;
   1:  PR[91,3] = PR[90,3] + 65.888;
   1:L PR[91] R[100]mm/sec CNT100;
   1:  PR[91,1] = PR[90,1] + 78.023;
   1:  PR[91,2] = PR[90,2] + -5.748;
   1:  PR[91,3] = PR[90,3] + 65.908;
   1:L PR[91] R[100]mm/sec CNT100;
   1:  PR[91,1] = PR[90,1] + 78.523;
   1:  PR[91,2] = PR[90,2] + -1.956;
   1:  PR[91,3] = PR[90,3] + 65.926;
   1:L PR[91] R[100]mm/sec CNT100;
   1:  PR[91,1] = PR[90,1] + 78.725;
   1:  PR[91,2] = PR[90,2] + -0.700;
   1:  PR[91,3] = PR[90,3] + 65.940;
   1:L PR[91] R[100]mm/sec CNT100;
   1:  PR[91,1] = PR[90,1] + 78.326;
   1:  PR[91,2] = PR[90,2] + 2.359;
   1:  PR[91,3] = PR[90,3] + 65.944;
   1:L PR[91] R[100]mm/sec CNT100;
   1:  PR[91,1] = PR[90,1] + 78.218;
   1:  PR[91,2] = PR[90,2] + 2.785;
   1:  PR[91,3] = PR[90,3] + 65.955;
   1:L PR[91] R[100]mm/sec CNT100;
   1:  PR[91,1] = PR[90,1] + 78.021;
   1:  PR[91,2] = PR[90,2] + 4.296;
   1:  PR[91,3] = PR[90,3] + 65.957;
   1:L PR[91] R[100]mm/sec CNT100;
   1:  PR[91,1] = PR[90,1] + 76.057;
   1:  PR[91,2] = PR[90,2] + 9.183;
   1:  PR[91,3] = PR[90,3] + 65.962;
   1:L PR[91] R[100]mm/sec CNT100;
   1:  PR[91,1] = PR[90,1] + 72.779;
   1:  PR[91,2] = PR[90,2] + 13.767;
   1:  PR[91,3] = PR[90,3] + 65.981;
   1:L PR[91] R[100]mm/sec CNT100;
   1:  PR[91,1] = PR[90,1] + 68.210;
   1:  PR[91,2] = PR[90,2] + 17.857;
   1:  PR[91,3] = PR[90,3] + 66.001;
   1:L PR[91] R[100]mm/sec CNT100;
   1:  PR[91,1] = PR[90,1] + 66.535;
   1:  PR[91,2] = PR[90,2] + 18.836;
   1:  PR[91,3] = PR[90,3] + 66.022;
   1:L PR[91] R[100]mm/sec CNT100;
   1:  PR[91,1] = PR[90,1] + 62.978;
   1:  PR[91,2] = PR[90,2] + 20.764;
   1:  PR[91,3] = PR[90,3] + 66.029;
   1:L PR[91] R[100]mm/sec CNT100;
   1:  PR[91,1] = PR[90,1] + 61.800;
   1:  PR[91,2] = PR[90,2] + 21.308;
   1:  PR[91,3] = PR[90,3] + 66.043;
   1:L PR[91] R[100]mm/sec CNT100;
   1:  PR[91,1] = PR[90,1] + 55.390;
   1:  PR[91,2] = PR[90,2] + 23.394;
   1:  PR[91,3] = PR[90,3] + 66.048;
   1:L PR[91] R[100]mm/sec CNT100;
   1:  PR[91,1] = PR[90,1] + 50.424;
   1:  PR[91,2] = PR[90,2] + 24.318;
   1:  PR[91,3] = PR[90,3] + 66.072;
   1:L PR[91] R[100]mm/sec CNT100;
   1:  PR[91,1] = PR[90,1] + 46.538;
   1:  PR[91,2] = PR[90,2] + 24.674;
   1:  PR[91,3] = PR[90,3] + 66.090;
   1:L PR[91] R[100]mm/sec CNT100;
   1:  PR[91,1] = PR[90,1] + 45.797;
   1:  PR[91,2] = PR[90,2] + 24.763;
   1:  PR[91,3] = PR[90,3] + 66.103;
   1:L PR[91] R[100]mm/sec CNT100;
   1:  PR[91,1] = PR[90,1] + 40.204;
   1:  PR[91,2] = PR[90,2] + 24.749;
   1:  PR[91,3] = PR[90,3] + 66.106;
   1:L PR[91] R[100]mm/sec CNT100;
   1:  PR[91,1] = PR[90,1] + 34.276;
   1:  PR[91,2] = PR[90,2] + 23.988;
   1:  PR[91,3] = PR[90,3] + 66.126;
   1:L PR[91] R[100]mm/sec CNT100;
   1:  PR[91,1] = PR[90,1] + 32.821;
   1:  PR[91,2] = PR[90,2] + 23.601;
   1:  PR[91,3] = PR[90,3] + 66.147;
   1:L PR[91] R[100]mm/sec CNT100;
   1:  PR[91,1] = PR[90,1] + 29.186;
   1:  PR[91,2] = PR[90,2] + 22.572;
   1:  PR[91,3] = PR[90,3] + 66.152;
   1:L PR[91] R[100]mm/sec CNT100;
   1:  PR[91,1] = PR[90,1] + 28.119;
   1:  PR[91,2] = PR[90,2] + 22.830;
   1:  PR[91,3] = PR[90,3] + 66.166;
   1:L PR[91] R[100]mm/sec CNT100;
   1:  PR[91,1] = PR[90,1] + 22.787;
   1:  PR[91,2] = PR[90,2] + 23.828;
   1:  PR[91,3] = PR[90,3] + 66.170;
   1:L PR[91] R[100]mm/sec CNT100;
   1:  PR[91,1] = PR[90,1] + 17.169;
   1:  PR[91,2] = PR[90,2] + 23.601;
   1:  PR[91,3] = PR[90,3] + 66.189;
   1:L PR[91] R[100]mm/sec CNT100;
   1:  PR[91,1] = PR[90,1] + 17.141;
   1:  PR[91,2] = PR[90,2] + 23.595;
   1:  PR[91,3] = PR[90,3] + 66.209;
   1:L PR[91] R[100]mm/sec CNT100;
   1:  PR[91,1] = PR[90,1] + 11.740;
   1:  PR[91,2] = PR[90,2] + 22.123;
   1:L PR[91] R[100]mm/sec CNT100;
   1:  PR[91,1] = PR[90,1] + 10.925;
   1:  PR[91,2] = PR[90,2] + 21.749;
   1:  PR[91,3] = PR[90,3] + 66.228;
   1:L PR[91] R[100]mm/sec CNT100;
   1:  PR[91,1] = PR[90,1] + 6.439;
   1:  PR[91,2] = PR[90,2] + 19.396;
   1:  PR[91,3] = PR[90,3] + 66.232;
   1:L PR[91] R[100]mm/sec CNT100;
   1:  PR[91,1] = PR[90,1] + 4.247;
   1:  PR[91,2] = PR[90,2] + 20.429;
   1:  PR[91,3] = PR[90,3] + 66.250;
   1:L PR[91] R[100]mm/sec CNT100;
   1:  PR[91,1] = PR[90,1] + 1.585;
   1:  PR[91,2] = PR[90,2] + 21.221;
   1:  PR[91,3] = PR[90,3] + 66.258;
   1:L PR[91] R[100]mm/sec CNT100;
   1:  PR[91,1] = PR[90,1] + -1.634;
   1:  PR[91,2] = PR[90,2] + 22.138;
   1:  PR[91,3] = PR[90,3] + 66.268;
   1:L PR[91] R[100]mm/sec CNT100;
   1:  PR[91,1] = PR[90,1] + -6.863;
   1:  PR[91,2] = PR[90,2] + 22.669;
   1:  PR[91,3] = PR[90,3] + 66.280;
   1:L PR[91] R[100]mm/sec CNT100;
   1:  PR[91,1] = PR[90,1] + -7.633;
   1:  PR[91,2] = PR[90,2] + 22.737;
   1:  PR[91,3] = PR[90,3] + 66.298;
   1:L PR[91] R[100]mm/sec CNT100;
   1:  PR[91,1] = PR[90,1] + -13.436;
   1:  PR[91,2] = PR[90,2] + 22.282;
   1:  PR[91,3] = PR[90,3] + 66.301;
   1:L PR[91] R[100]mm/sec CNT100;
   1:  PR[91,1] = PR[90,1] + -17.195;
   1:  PR[91,2] = PR[90,2] + 21.281;
   1:  PR[91,3] = PR[90,3] + 66.322;
   1:L PR[91] R[100]mm/sec CNT100;
   1:  PR[91,1] = PR[90,1] + -18.805;
   1:  PR[91,2] = PR[90,2] + 20.815;
   1:  PR[91,3] = PR[90,3] + 66.335;
   1:L PR[91] R[100]mm/sec CNT100;
   1:  PR[91,1] = PR[90,1] + -21.649;
   1:  PR[91,2] = PR[90,2] + 19.594;
   1:  PR[91,3] = PR[90,3] + 66.341;
   1:L PR[91] R[100]mm/sec CNT100;
   1:  PR[91,1] = PR[90,1] + -24.288;
   1:  PR[91,2] = PR[90,2] + 20.090;
   1:  PR[91,3] = PR[90,3] + 66.352;
   1:L PR[91] R[100]mm/sec CNT100;
   1:  PR[91,1] = PR[90,1] + -27.907;
   1:  PR[91,2] = PR[90,2] + 20.917;
   1:  PR[91,3] = PR[90,3] + 66.362;
   1:L PR[91] R[100]mm/sec CNT100;
   1:  PR[91,1] = PR[90,1] + -32.708;
   1:  PR[91,2] = PR[90,2] + 21.532;
   1:  PR[91,3] = PR[90,3] + 66.375;
   1:L PR[91] R[100]mm/sec CNT100;
   1:  PR[91,1] = PR[90,1] + -35.331;
   1:  PR[91,2] = PR[90,2] + 22.030;
   1:  PR[91,3] = PR[90,3] + 66.392;
   1:L PR[91] R[100]mm/sec CNT100;
   1:  PR[91,1] = PR[90,1] + -41.612;
   1:  PR[91,2] = PR[90,2] + 22.556;
   1:  PR[91,3] = PR[90,3] + 66.401;
   1:L PR[91] R[100]mm/sec CNT100;
   1:  PR[91,1] = PR[90,1] + -42.021;
   1:  PR[91,2] = PR[90,2] + 22.579;
   1:  PR[91,3] = PR[90,3] + 66.424;
   1:L PR[91] R[100]mm/sec CNT100;
   1:  PR[91,1] = PR[90,1] + -47.406;
   1:  PR[91,2] = PR[90,2] + 22.482;
   1:  PR[91,3] = PR[90,3] + 66.425;
   1:L PR[91] R[100]mm/sec CNT100;
   1:  PR[91,1] = PR[90,1] + -51.766;
   1:  PR[91,2] = PR[90,2] + 22.211;
   1:  PR[91,3] = PR[90,3] + 66.444;
   1:L PR[91] R[100]mm/sec CNT100;
   1:  PR[91,1] = PR[90,1] + -52.482;
   1:  PR[91,2] = PR[90,2] + 22.093;
   1:  PR[91,3] = PR[90,3] + 66.460;
   1:L PR[91] R[100]mm/sec CNT100;
   1:  PR[91,1] = PR[90,1] + -53.591;
   1:  PR[91,2] = PR[90,2] + 21.865;
   1:  PR[91,3] = PR[90,3] + 66.462;
   1:L PR[91] R[100]mm/sec CNT100;
   1:  PR[91,1] = PR[90,1] + -57.222;
   1:  PR[91,2] = PR[90,2] + 21.096;
   1:  PR[91,3] = PR[90,3] + 66.466;
   1:L PR[91] R[100]mm/sec CNT100;
   1:  PR[91,1] = PR[90,1] + -58.947;
   1:  PR[91,2] = PR[90,2] + 20.713;
   1:  PR[91,3] = PR[90,3] + 66.479;
   1:L PR[91] R[100]mm/sec CNT100;
   1:  PR[91,1] = PR[90,1] + -61.458;
   1:  PR[91,2] = PR[90,2] + 19.734;
   1:  PR[91,3] = PR[90,3] + 66.485;
   1:L PR[91] R[100]mm/sec CNT100;
   1:  PR[91] = PR[90];
   1:  PR[91,1] = PR[90,1] + -63.810;
   1:  PR[91,2] = PR[90,2] + 18.535;
   1:  PR[91,3] = PR[90,3] + 67.795;
   1:L PR[91] R[100]mm/sec CNT100;
   1:  PR[91,1] = PR[90,1] + -68.859;
   1:  PR[91,2] = PR[90,2] + 15.436;
   1:  PR[91,3] = PR[90,3] + 66.505;
   1:L PR[91] R[100]mm/sec CNT100;
   1:  PR[91,1] = PR[90,1] + -69.033;
   1:  PR[91,2] = PR[90,2] + 15.277;
   1:  PR[91,3] = PR[90,3] + 66.527;
   1:L PR[91] R[100]mm/sec CNT100;
   1:  PR[91,1] = PR[90,1] + -72.471;
   1:  PR[91,2] = PR[90,2] + 11.875;
   1:L PR[91] R[100]mm/sec CNT100;
   1:  PR[91,1] = PR[90,1] + -75.094;
   1:  PR[91,2] = PR[90,2] + 7.877;
   1:  PR[91,3] = PR[90,3] + 66.545;
   1:L PR[91] R[100]mm/sec CNT100;
   1:  PR[91,1] = PR[90,1] + -76.669;
   1:  PR[91,2] = PR[90,2] + 3.632;
   1:  PR[91,3] = PR[90,3] + 66.562;
   1:L PR[91] R[100]mm/sec CNT100;
   1:  PR[91,1] = PR[90,1] + -76.910;
   1:  PR[91,2] = PR[90,2] + 1.632;
   1:  PR[91,3] = PR[90,3] + 66.578;
   1:L PR[91] R[100]mm/sec CNT100;
   1:  PR[91,1] = PR[90,1] + -77.335;
   1:  PR[91,2] = PR[90,2] + -0.735;
   1:  PR[91,3] = PR[90,3] + 66.585;
   1:L PR[91] R[100]mm/sec CNT100;
   1:  PR[91,1] = PR[90,1] + -76.778;
   1:  PR[91,2] = PR[90,2] + -5.303;
   1:  PR[91,3] = PR[90,3] + 66.594;
   1:L PR[91] R[100]mm/sec CNT100;
   1:  PR[91,1] = PR[90,1] + -76.677;
   1:  PR[91,2] = PR[90,2] + -5.570;
   1:  PR[91,3] = PR[90,3] + 66.610;
   1:L PR[91] R[100]mm/sec CNT100;
   1:  PR[91,1] = PR[90,1] + -75.006;
   1:  PR[91,2] = PR[90,2] + -9.676;
   1:  PR[91,3] = PR[90,3] + 66.611;
   1:L PR[91] R[100]mm/sec CNT100;
   1:  PR[91,1] = PR[90,1] + -74.815;
   1:  PR[91,2] = PR[90,2] + -9.945;
   1:  PR[91,3] = PR[90,3] + 66.627;
   1:L PR[91] R[100]mm/sec CNT100;
   1:  PR[91,1] = PR[90,1] + -72.047;
   1:  PR[91,2] = PR[90,2] + -13.778;
   1:  PR[91,3] = PR[90,3] + 66.628;
   1:L PR[91] R[100]mm/sec CNT100;
   1:  PR[91,1] = PR[90,1] + -70.805;
   1:  PR[91,2] = PR[90,2] + -14.904;
   1:  PR[91,3] = PR[90,3] + 66.645;
   1:L PR[91] R[100]mm/sec CNT100;
   1:  PR[91,1] = PR[90,1] + -67.995;
   1:  PR[91,2] = PR[90,2] + -17.410;
   1:  PR[91,3] = PR[90,3] + 66.651;
   1:L PR[91] R[100]mm/sec CNT100;
   1:  PR[91,1] = PR[90,1] + -64.532;
   1:  PR[91,2] = PR[90,2] + -19.486;
   1:  PR[91,3] = PR[90,3] + 66.664;
   1:L PR[91] R[100]mm/sec CNT100;
   1:  PR[91,1] = PR[90,1] + -62.972;
   1:  PR[91,2] = PR[90,2] + -20.403;
   1:  PR[91,3] = PR[90,3] + 66.679;
   1:L PR[91] R[100]mm/sec CNT100;
   1:  PR[91,1] = PR[90,1] + -59.253;
   1:  PR[91,2] = PR[90,2] + -21.797;
   1:  PR[91,3] = PR[90,3] + 66.685;
   1:L PR[91] R[100]mm/sec CNT100;
   1:  PR[91,1] = PR[90,1] + -57.193;
   1:  PR[91,2] = PR[90,2] + -22.531;
   1:  PR[91,3] = PR[90,3] + 66.699;
   1:L PR[91] R[100]mm/sec CNT100;
   1:  PR[91,1] = PR[90,1] + -55.921;
   1:  PR[91,2] = PR[90,2] + -22.838;
   1:  PR[91,3] = PR[90,3] + 66.707;
   1:L PR[91] R[100]mm/sec CNT100;
   1:  PR[91,1] = PR[90,1] + -51.334;
   1:  PR[91,2] = PR[90,2] + -23.715;
   1:  PR[91,3] = PR[90,3] + 66.712;
   1:L PR[91] R[100]mm/sec CNT100;
   1:  PR[91,1] = PR[90,1] + -45.448;
   1:  PR[91,2] = PR[90,2] + -24.278;
   1:  PR[91,3] = PR[90,3] + 66.728;
   1:L PR[91] R[100]mm/sec CNT100;
   1:  PR[91,1] = PR[90,1] + -39.961;
   1:  PR[91,2] = PR[90,2] + -24.196;
   1:  PR[91,3] = PR[90,3] + 66.750;
   1:L PR[91] R[100]mm/sec CNT100;
   1:  PR[91,1] = PR[90,1] + -34.145;
   1:  PR[91,2] = PR[90,2] + -23.855;
   1:  PR[91,3] = PR[90,3] + 66.769;
   1:L PR[91] R[100]mm/sec CNT100;
   1:  PR[91,1] = PR[90,1] + -26.197;
   1:  PR[91,2] = PR[90,2] + -22.780;
   1:  PR[91,3] = PR[90,3] + 66.790;
   1:L PR[91] R[100]mm/sec CNT100;
   1:  PR[91,1] = PR[90,1] + -24.938;
   1:  PR[91,2] = PR[90,2] + -22.490;
   1:  PR[91,3] = PR[90,3] + 66.819;
   1:L PR[91] R[100]mm/sec CNT100;
   1:  PR[91,1] = PR[90,1] + -20.205;
   1:  PR[91,2] = PR[90,2] + -21.602;
   1:  PR[91,3] = PR[90,3] + 66.823;
   1:L PR[91] R[100]mm/sec CNT100;
   1:  PR[91,1] = PR[90,1] + -18.135;
   1:  PR[91,2] = PR[90,2] + -22.490;
   1:  PR[91,3] = PR[90,3] + 66.840;
   1:L PR[91] R[100]mm/sec CNT100;
   1:  PR[91,1] = PR[90,1] + -17.081;
   1:  PR[91,2] = PR[90,2] + -22.797;
   1:  PR[91,3] = PR[90,3] + 66.848;
   1:L PR[91] R[100]mm/sec CNT100;
   1:  PR[91,1] = PR[90,1] + -12.784;
   1:  PR[91,2] = PR[90,2] + -23.942;
   1:  PR[91,3] = PR[90,3] + 66.852;
   1:L PR[91] R[100]mm/sec CNT100;
   1:  PR[91,1] = PR[90,1] + -6.886;
   1:  PR[91,2] = PR[90,2] + -24.417;
   1:  PR[91,3] = PR[90,3] + 66.868;
   1:L PR[91] R[100]mm/sec CNT100;
   1:  PR[91,1] = PR[90,1] + -4.888;
   1:  PR[91,2] = PR[90,2] + -24.242;
   1:  PR[91,3] = PR[90,3] + 66.889;
   1:L PR[91] R[100]mm/sec CNT100;
   1:  PR[91,1] = PR[90,1] + -0.830;
   1:  PR[91,2] = PR[90,2] + -23.832;
   1:  PR[91,3] = PR[90,3] + 66.896;
   1:L PR[91] R[100]mm/sec CNT100;
   1:  PR[91,1] = PR[90,1] + 3.704;
   1:  PR[91,2] = PR[90,2] + -22.542;
   1:  PR[91,3] = PR[90,3] + 66.911;
   1:L PR[91] R[100]mm/sec CNT100;
   1:  PR[91,1] = PR[90,1] + 5.146;
   1:  PR[91,2] = PR[90,2] + -22.114;
   1:  PR[91,3] = PR[90,3] + 66.928;
   1:L PR[91] R[100]mm/sec CNT100;
   1:  PR[91,1] = PR[90,1] + 6.737;
   1:  PR[91,2] = PR[90,2] + -21.344;
   1:  PR[91,3] = PR[90,3] + 66.933;
   1:L PR[91] R[100]mm/sec CNT100;
   1:  PR[91,1] = PR[90,1] + 9.661;
   1:  PR[91,2] = PR[90,2] + -22.900;
   1:  PR[91,3] = PR[90,3] + 66.939;
   1:L PR[91] R[100]mm/sec CNT100;
   1:  PR[91,1] = PR[90,1] + 11.608;
   1:  PR[91,2] = PR[90,2] + -23.794;
   1:  PR[91,3] = PR[90,3] + 66.951;
   1:L PR[91] R[100]mm/sec CNT100;
   1:  PR[91,1] = PR[90,1] + 16.445;
   1:  PR[91,2] = PR[90,2] + -25.112;
   1:  PR[91,3] = PR[90,3] + 66.959;
   1:L PR[91] R[100]mm/sec CNT100;
   1:  PR[91,1] = PR[90,1] + 17.133;
   1:  PR[91,2] = PR[90,2] + -25.261;
   1:  PR[91,3] = PR[90,3] + 66.977;
   1:L PR[91] R[100]mm/sec CNT100;
   1:  PR[91,1] = PR[90,1] + 22.417;
   1:  PR[91,2] = PR[90,2] + -25.475;
   1:  PR[91,3] = PR[90,3] + 66.979;
   1:L PR[91] R[100]mm/sec CNT100;
   1:  PR[91,1] = PR[90,1] + 22.776;
   1:  PR[91,2] = PR[90,2] + -25.463;
   1:  PR[91,3] = PR[90,3] + 66.998;
   1:L PR[91] R[100]mm/sec CNT100;
   1:  PR[91,1] = PR[90,1] + 23.448;
   1:  PR[91,2] = PR[90,2] + -25.361;
   1:  PR[91,3] = PR[90,3] + 66.999;
   1:L PR[91] R[100]mm/sec CNT100;
   1:  PR[91,1] = PR[90,1] + 28.677;
   1:  PR[91,2] = PR[90,2] + -24.373;
   1:  PR[91,3] = PR[90,3] + 67.002;
   1:L PR[91] R[100]mm/sec CNT100;
   1:  PR[91,1] = PR[90,1] + 32.404;
   1:  PR[91,2] = PR[90,2] + -25.394;
   1:  PR[91,3] = PR[90,3] + 67.021;
   1:L PR[91] R[100]mm/sec CNT100;
   1:  PR[91,1] = PR[90,1] + 33.782;
   1:  PR[91,2] = PR[90,2] + -25.725;
   1:  PR[91,3] = PR[90,3] + 67.035;
   1:L PR[91] R[100]mm/sec CNT100;
   1:  PR[91,1] = PR[90,1] + 36.461;
   1:  PR[91,2] = PR[90,2] + -26.096;
   1:  PR[91,3] = PR[90,3] + 67.040;
   1:L PR[91] R[100]mm/sec CNT100;
   1:  PR[91,1] = PR[90,1] + 39.078;
   1:  PR[91,2] = PR[90,2] + -26.428;
   1:  PR[91,3] = PR[90,3] + 67.049;
   1:L PR[91] R[100]mm/sec CNT100;
   1:  PR[91,1] = PR[90,1] + 41.361;
   1:  PR[91,2] = PR[90,2] + -26.437;
   1:  PR[91,3] = PR[90,3] + 67.059;
   1:L PR[91] R[100]mm/sec CNT100;
   1:  PR[91,1] = PR[90,1] + 44.834;
   1:  PR[91,2] = PR[90,2] + -26.423;
   1:  PR[91,3] = PR[90,3] + 67.067;
   1:L PR[91] R[100]mm/sec CNT100;
   1:  PR[91,1] = PR[90,1] + 47.733;
   1:  PR[91,2] = PR[90,2] + -26.075;
   1:  PR[91,3] = PR[90,3] + 67.079;
   1:L PR[91] R[100]mm/sec CNT100;
   1:  PR[91,1] = PR[90,1] + 49.754;
   1:  PR[91,2] = PR[90,2] + -25.890;
   1:  PR[91,3] = PR[90,3] + 67.090;
   1:L PR[91] R[100]mm/sec CNT100;
   1:  PR[91,1] = PR[90,1] + 54.334;
   1:  PR[91,2] = PR[90,2] + -25.031;
   1:  PR[91,3] = PR[90,3] + 67.097;
   1:L PR[91] R[100]mm/sec CNT100;
   1:  PR[91,1] = PR[90,1] + 60.421;
   1:  PR[91,2] = PR[90,2] + -23.054;
   1:  PR[91,3] = PR[90,3] + 67.113;
   1:L PR[91] R[100]mm/sec CNT100;
   1:  PR[91,1] = PR[90,1] + 62.374;
   1:  PR[91,2] = PR[90,2] + -22.151;
   1:  PR[91,3] = PR[90,3] + 67.136;
   1:L PR[91] R[100]mm/sec CNT100;
   1:  PR[91,1] = PR[90,1] + 67.314;
   1:  PR[91,2] = PR[90,2] + -19.477;
   1:  PR[91,3] = PR[90,3] + 67.144;
   1:L PR[91] R[100]mm/sec CNT100;
   1:  PR[91,1] = PR[90,1] + 67.332;
   1:  PR[91,2] = PR[90,2] + -19.466;
   1:  PR[91,3] = PR[90,3] + 67.164;
   1:L PR[91] R[100]mm/sec CNT100;
   1:  PR[91,1] = PR[90,1] + 67.721;
   1:  PR[91,2] = PR[90,2] + -19.145;
   1:L PR[91] R[100]mm/sec CNT100;
   1:  PR[91,1] = PR[90,1] + 71.945;
   1:  PR[91,2] = PR[90,2] + -15.369;
   1:  PR[91,3] = PR[90,3] + 67.166;
   1:L PR[91] R[100]mm/sec CNT100;
   1:  PR[91,1] = PR[90,1] + 75.261;
   1:  PR[91,2] = PR[90,2] + -10.736;
   1:  PR[91,3] = PR[90,3] + 67.186;
   1:L PR[91] R[100]mm/sec CNT100;
   1:  PR[91,1] = PR[90,1] + 77.245;
   1:  PR[91,2] = PR[90,2] + -5.799;
   1:  PR[91,3] = PR[90,3] + 67.206;
   1:L PR[91] R[100]mm/sec CNT100;
   1:  PR[91,1] = PR[90,1] + 77.648;
   1:  PR[91,2] = PR[90,2] + -2.743;
   1:  PR[91,3] = PR[90,3] + 67.225;
   1:L PR[91] R[100]mm/sec CNT100;
   1:  PR[91,1] = PR[90,1] + 77.976;
   1:  PR[91,2] = PR[90,2] + -0.700;
   1:  PR[91,3] = PR[90,3] + 67.236;
   1:L PR[91] R[100]mm/sec CNT100;
   1:  PR[91,1] = PR[90,1] + 77.688;
   1:  PR[91,2] = PR[90,2] + 1.503;
   1:  PR[91,3] = PR[90,3] + 67.244;
   1:L PR[91] R[100]mm/sec CNT100;
   1:  PR[91,1] = PR[90,1] + 77.534;
   1:  PR[91,2] = PR[90,2] + 2.116;
   1:  PR[91,3] = PR[90,3] + 67.252;
   1:L PR[91] R[100]mm/sec CNT100;
   1:  PR[91,1] = PR[90,1] + 77.243;
   1:  PR[91,2] = PR[90,2] + 4.345;
   1:  PR[91,3] = PR[90,3] + 67.254;
   1:L PR[91] R[100]mm/sec CNT100;
   1:  PR[91,1] = PR[90,1] + 75.259;
   1:  PR[91,2] = PR[90,2] + 9.281;
   1:  PR[91,3] = PR[90,3] + 67.262;
   1:L PR[91] R[100]mm/sec CNT100;
   1:  PR[91,1] = PR[90,1] + 71.946;
   1:  PR[91,2] = PR[90,2] + 13.909;
   1:  PR[91,3] = PR[90,3] + 67.281;
   1:L PR[91] R[100]mm/sec CNT100;
   1:  PR[91,1] = PR[90,1] + 67.720;
   1:  PR[91,2] = PR[90,2] + 17.689;
   1:  PR[91,3] = PR[90,3] + 67.301;
   1:L PR[91] R[100]mm/sec CNT100;
   1:  PR[91,1] = PR[90,1] + 67.345;
   1:  PR[91,2] = PR[90,2] + 17.999;
   1:  PR[91,3] = PR[90,3] + 67.321;
   1:L PR[91] R[100]mm/sec CNT100;
   1:  PR[91,1] = PR[90,1] + 67.331;
   1:  PR[91,2] = PR[90,2] + 18.007;
   1:  PR[91,3] = PR[90,3] + 67.323;
   1:L PR[91] R[100]mm/sec CNT100;
   1:  PR[91,1] = PR[90,1] + 62.385;
   1:  PR[91,2] = PR[90,2] + 20.688;
   1:L PR[91] R[100]mm/sec CNT100;
   1:  PR[91,1] = PR[90,1] + 60.433;
   1:  PR[91,2] = PR[90,2] + 21.590;
   1:  PR[91,3] = PR[90,3] + 67.343;
   1:L PR[91] R[100]mm/sec CNT100;
   1:  PR[91,1] = PR[90,1] + 54.335;
   1:  PR[91,2] = PR[90,2] + 23.572;
   1:  PR[91,3] = PR[90,3] + 67.351;
   1:L PR[91] R[100]mm/sec CNT100;
   1:  PR[91,1] = PR[90,1] + 49.754;
   1:  PR[91,2] = PR[90,2] + 24.431;
   1:  PR[91,3] = PR[90,3] + 67.374;
   1:L PR[91] R[100]mm/sec CNT100;
   1:  PR[91,1] = PR[90,1] + 47.733;
   1:  PR[91,2] = PR[90,2] + 24.616;
   1:  PR[91,3] = PR[90,3] + 67.391;
   1:L PR[91] R[100]mm/sec CNT100;
   1:  PR[91,1] = PR[90,1] + 44.834;
   1:  PR[91,2] = PR[90,2] + 24.964;
   1:  PR[91,3] = PR[90,3] + 67.398;
   1:L PR[91] R[100]mm/sec CNT100;
   1:  PR[91,1] = PR[90,1] + 41.361;
   1:  PR[91,2] = PR[90,2] + 24.978;
   1:  PR[91,3] = PR[90,3] + 67.408;
   1:L PR[91] R[100]mm/sec CNT100;
   1:  PR[91,1] = PR[90,1] + 39.078;
   1:  PR[91,2] = PR[90,2] + 24.969;
   1:  PR[91,3] = PR[90,3] + 67.421;
   1:L PR[91] R[100]mm/sec CNT100;
   1:  PR[91,1] = PR[90,1] + 36.461;
   1:  PR[91,2] = PR[90,2] + 24.637;
   1:  PR[91,3] = PR[90,3] + 67.429;
   1:L PR[91] R[100]mm/sec CNT100;
   1:  PR[91,1] = PR[90,1] + 33.782;
   1:  PR[91,2] = PR[90,2] + 24.266;
   1:  PR[91,3] = PR[90,3] + 67.438;
   1:L PR[91] R[100]mm/sec CNT100;
   1:  PR[91,1] = PR[90,1] + 32.404;
   1:  PR[91,2] = PR[90,2] + 23.935;
   1:  PR[91,3] = PR[90,3] + 67.448;
   1:L PR[91] R[100]mm/sec CNT100;
   1:  PR[91,1] = PR[90,1] + 28.677;
   1:  PR[91,2] = PR[90,2] + 22.915;
   1:  PR[91,3] = PR[90,3] + 67.453;
   1:L PR[91] R[100]mm/sec CNT100;
   1:  PR[91,1] = PR[90,1] + 23.448;
   1:  PR[91,2] = PR[90,2] + 23.902;
   1:  PR[91,3] = PR[90,3] + 67.467;
   1:L PR[91] R[100]mm/sec CNT100;
   1:  PR[91,1] = PR[90,1] + 22.770;
   1:  PR[91,2] = PR[90,2] + 24.005;
   1:  PR[91,3] = PR[90,3] + 67.486;
   1:L PR[91] R[100]mm/sec CNT100;
   1:  PR[91,1] = PR[90,1] + 22.416;
   1:  PR[91,2] = PR[90,2] + 24.016;
   1:  PR[91,3] = PR[90,3] + 67.488;
   1:L PR[91] R[100]mm/sec CNT100;
   1:  PR[91,1] = PR[90,1] + 17.132;
   1:  PR[91,2] = PR[90,2] + 23.802;
   1:  PR[91,3] = PR[90,3] + 67.489;
   1:L PR[91] R[100]mm/sec CNT100;
   1:  PR[91,1] = PR[90,1] + 16.443;
   1:  PR[91,2] = PR[90,2] + 23.653;
   1:  PR[91,3] = PR[90,3] + 67.508;
   1:L PR[91] R[100]mm/sec CNT100;
   1:  PR[91,1] = PR[90,1] + 11.606;
   1:  PR[91,2] = PR[90,2] + 22.335;
   1:  PR[91,3] = PR[90,3] + 67.511;
   1:L PR[91] R[100]mm/sec CNT100;
   1:  PR[91,1] = PR[90,1] + 9.668;
   1:  PR[91,2] = PR[90,2] + 21.446;
   1:  PR[91,3] = PR[90,3] + 67.529;
   1:L PR[91] R[100]mm/sec CNT100;
   1:  PR[91,1] = PR[90,1] + 6.734;
   1:  PR[91,2] = PR[90,2] + 19.917;
   1:  PR[91,3] = PR[90,3] + 67.536;
   1:L PR[91] R[100]mm/sec CNT100;
   1:  PR[91,1] = PR[90,1] + 5.155;
   1:  PR[91,2] = PR[90,2] + 20.653;
   1:  PR[91,3] = PR[90,3] + 67.548;
   1:L PR[91] R[100]mm/sec CNT100;
   1:  PR[91,1] = PR[90,1] + 3.687;
   1:  PR[91,2] = PR[90,2] + 21.090;
   1:  PR[91,3] = PR[90,3] + 67.554;
   1:L PR[91] R[100]mm/sec CNT100;
   1:  PR[91,1] = PR[90,1] + -0.800;
   1:  PR[91,2] = PR[90,2] + 22.367;
   1:  PR[91,3] = PR[90,3] + 67.560;
   1:L PR[91] R[100]mm/sec CNT100;
   1:  PR[91,1] = PR[90,1] + -4.857;
   1:  PR[91,2] = PR[90,2] + 22.780;
   1:  PR[91,3] = PR[90,3] + 67.576;
   1:L PR[91] R[100]mm/sec CNT100;
   1:  PR[91,1] = PR[90,1] + -6.872;
   1:  PR[91,2] = PR[90,2] + 22.958;
   1:  PR[91,3] = PR[90,3] + 67.591;
   1:L PR[91] R[100]mm/sec CNT100;
   1:  PR[91,1] = PR[90,1] + -12.776;
   1:  PR[91,2] = PR[90,2] + 22.484;
   1:  PR[91,3] = PR[90,3] + 67.598;
   1:L PR[91] R[100]mm/sec CNT100;
   1:  PR[91,1] = PR[90,1] + -17.078;
   1:  PR[91,2] = PR[90,2] + 21.338;
   1:  PR[91,3] = PR[90,3] + 67.619;
   1:L PR[91] R[100]mm/sec CNT100;
   1:  PR[91,1] = PR[90,1] + -18.128;
   1:  PR[91,2] = PR[90,2] + 21.034;
   1:  PR[91,3] = PR[90,3] + 67.635;
   1:L PR[91] R[100]mm/sec CNT100;
   1:  PR[91,1] = PR[90,1] + -20.205;
   1:  PR[91,2] = PR[90,2] + 20.143;
   1:  PR[91,3] = PR[90,3] + 67.639;
   1:L PR[91] R[100]mm/sec CNT100;
   1:  PR[91,1] = PR[90,1] + -24.937;
   1:  PR[91,2] = PR[90,2] + 21.031;
   1:  PR[91,3] = PR[90,3] + 67.647;
   1:L PR[91] R[100]mm/sec CNT100;
   1:  PR[91,1] = PR[90,1] + -26.224;
   1:  PR[91,2] = PR[90,2] + 21.326;
   1:  PR[91,3] = PR[90,3] + 67.664;
   1:L PR[91] R[100]mm/sec CNT100;
   1:  PR[91,1] = PR[90,1] + -33.547;
   1:  PR[91,2] = PR[90,2] + 22.264;
   1:  PR[91,3] = PR[90,3] + 67.669;
   1:L PR[91] R[100]mm/sec CNT100;
   1:  PR[91,1] = PR[90,1] + -34.277;
   1:  PR[91,2] = PR[90,2] + 22.402;
   1:  PR[91,3] = PR[90,3] + 67.695;
   1:L PR[91] R[100]mm/sec CNT100;
   1:  PR[91,1] = PR[90,1] + -36.007;
   1:  PR[91,2] = PR[90,2] + 22.547;
   1:  PR[91,3] = PR[90,3] + 67.698;
   1:L PR[91] R[100]mm/sec CNT100;
   1:  PR[91,1] = PR[90,1] + -40.912;
   1:  PR[91,2] = PR[90,2] + 22.827;
   1:  PR[91,3] = PR[90,3] + 67.704;
   1:L PR[91] R[100]mm/sec CNT100;
   1:  PR[91,1] = PR[90,1] + -43.221;
   1:  PR[91,2] = PR[90,2] + 22.726;
   1:  PR[91,3] = PR[90,3] + 67.722;
   1:L PR[91] R[100]mm/sec CNT100;
   1:  PR[91,1] = PR[90,1] + -46.877;
   1:  PR[91,2] = PR[90,2] + 22.665;
   1:  PR[91,3] = PR[90,3] + 67.730;
   1:L PR[91] R[100]mm/sec CNT100;
   1:  PR[91,1] = PR[90,1] + -49.875;
   1:  PR[91,2] = PR[90,2] + 22.478;
   1:  PR[91,3] = PR[90,3] + 67.743;
   1:L PR[91] R[100]mm/sec CNT100;
   1:  PR[91,1] = PR[90,1] + -51.957;
   1:  PR[91,2] = PR[90,2] + 22.134;
   1:  PR[91,3] = PR[90,3] + 67.754;
   1:L PR[91] R[100]mm/sec CNT100;
   1:  PR[91,1] = PR[90,1] + -54.908;
   1:  PR[91,2] = PR[90,2] + 21.528;
   1:  PR[91,3] = PR[90,3] + 67.761;
   1:L PR[91] R[100]mm/sec CNT100;
   1:  PR[91,1] = PR[90,1] + -57.775;
   1:  PR[91,2] = PR[90,2] + 20.911;
   1:  PR[91,3] = PR[90,3] + 67.772;
   1:L PR[91] R[100]mm/sec CNT100;
   1:  PR[91,1] = PR[90,1] + -61.096;
   1:  PR[91,2] = PR[90,2] + 19.617;
   1:  PR[91,3] = PR[90,3] + 67.782;
   1:L PR[91] R[100]mm/sec CNT100 TB   .50sec,CALL END_PUD;
   1:  DO[117:Laser Start]=OFF;
   1:  PR[92] = PR[91];
   1:  PR[92,3] = PR[92,3] + 50;
   1:J PR[92] 10% FINE;
   1:  WAIT   5.00(sec);
   1:  DO[119:Gas]=OFF;
   1:  CALL HOME_ALL;
/POS
/END
